FUNCTION_BLOCK CLIENT_3_2 (* Client with 3 inputs and 2 outputs, needed for HTTP *)
  (* Standard: 61499-2; Description: Copyright (c) 2024 Monika Wenger This program and the accompanying materials are made available under the terms of the Eclipse Public License 2.0 which is available at https://www.eclipse.org/legal/epl-2.0/ SPDX-License-Identifier: EPL-2.0 *)
  (* Version 1.0, 2024-02-26, Monika Wenger *)
  PACKAGE iec61499::net;
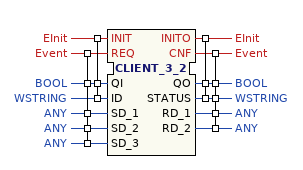
  EVENT_INPUT
    INIT : EInit WITH QI, ID; (* Open new connection (QI = TRUE) / Close connection (QI = FALSE) *)
    REQ WITH QI, SD_1, SD_2, SD_3; (* Transmits data to the server *)
  END_EVENT
  EVENT_OUTPUT
    INITO : EInit WITH QO, STATUS; (* New connection established (QI = TRUE) / connection closed (QI = FALSE) *)
    CNF WITH QO, STATUS, RD_1, RD_2; (* Response from the server *)
  END_EVENT
  VAR_INPUT
    QI : BOOL;
    ID : WSTRING;
    SD_1 : ANY; (* Token for authentication at the server *)
    SD_2 : ANY; (* Parameters for the message *)
    SD_3 : ANY; (* Body of the message *)
  END_VAR
  VAR_OUTPUT
    QO : BOOL;
    STATUS : WSTRING;
    RD_1 : ANY; (* Response code from the server *)
    RD_2 : ANY; (* Body from the server's response *)
  END_VAR
END_FUNCTION_BLOCK
